FUNCTION FC_Comms1 : INT
VAR_INPUT
	ix_gereed : BOOL;
	ix_ALARM : BOOL;
	//ix_bewegingVoltooid : BOOL;
END_VAR
VAR
END_VAR

// KUKA Robot naar PLC communicatie;

IF ix_gereed AND DB_PRG1.PRG1Stap = 60 AND NOT ix_ALARM THEN		//status beweging actief
	FC_Comms1 := 2;
ELSIF ix_gereed AND NOT ix_ALARM THEN								//status gereed wacht op beweeg
	FC_Comms1 := 1;
ELSIF ix_ALARM THEN													// status alarms
	FC_Comms1 := 4;
ELSE 
	FC_Comms1 := 3;													// iets anders 
END_IF

END_FUNCTION

(* stored: Version 1.1.0.1, ProductVersion 3.1.4024.12
   POU FC_Comms1: Id {16b8c8f8-ee1f-45bc-88d0-07396f66986f}, SpecialFunc None *)
